SYSTEM FLASHER10_TEST (* Test FLASHER10 with D10U10B service interface *)
  (* Standard: 61499-1; Classification: Communication; Function: Test; Type: DeviceNet *)
  (* Version 0.0, 2003-05-01, JHC, Rockwell Automation, Modified from D10U10B_TEST *)
  DEVICE HMI : FRAME_DEVICE
    RESOURCE INS : PANEL_RESOURCE
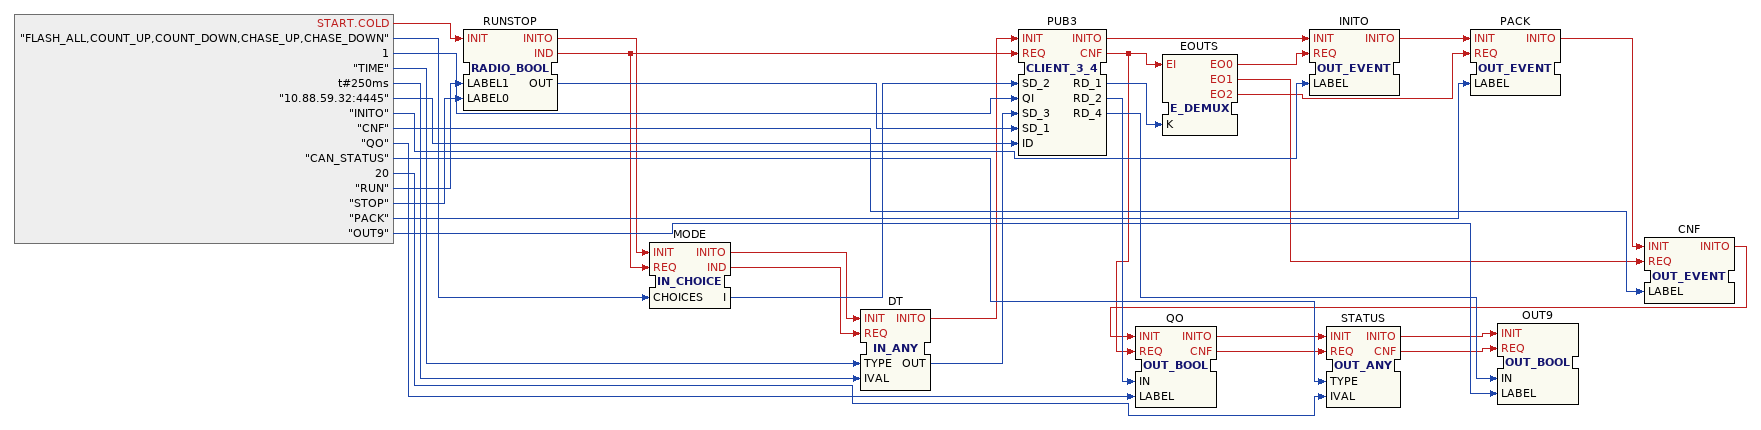
      FBS
        RUNSTOP : RADIO_BOOL;
        MODE : IN_CHOICE;
        DT : IN_ANY;
        PUB3 : CLIENT_3_4;
        EOUTS : E_DEMUX;
        INITO : OUT_EVENT;
        CNF : OUT_EVENT;
        QO : OUT_BOOL;
        STATUS : OUT_ANY;
        OUT9 : OUT_BOOL;
        PACK : OUT_EVENT;
      END_FBS
      EVENT_CONNECTIONS
        START.COLD TO RUNSTOP.INIT;
        RUNSTOP.INITO TO MODE.INIT;
        MODE.INITO TO DT.INIT;
        DT.INITO TO PUB3.INIT;
        PUB3.INITO TO INITO.INIT;
        INITO.INITO TO PACK.INIT;
        PACK.INITO TO CNF.INIT;
        CNF.INITO TO QO.INIT;
        QO.INITO TO STATUS.INIT;
        STATUS.INITO TO OUT9.INIT;
        RUNSTOP.IND TO MODE.REQ;
        MODE.IND TO DT.REQ;
        RUNSTOP.IND TO PUB3.REQ;
        PUB3.CNF TO QO.REQ;
        QO.CNF TO STATUS.REQ;
        STATUS.CNF TO OUT9.REQ;
        PUB3.CNF TO EOUTS.EI;
        EOUTS.EO0 TO INITO.REQ;
        EOUTS.EO1 TO CNF.REQ;
        EOUTS.EO2 TO PACK.REQ;
      END_CONNECTIONS
      DATA_CONNECTIONS
        MODE.I TO PUB3.SD_2;
        "FLASH_ALL,COUNT_UP,COUNT_DOWN,CHASE_UP,CHASE_DOWN" TO MODE.CHOICES;
        1 TO PUB3.QI;
        DT.OUT TO PUB3.SD_3;
        RUNSTOP.OUT TO PUB3.SD_1;
        PUB3.RD_1 TO EOUTS.K;
        PUB3.RD_2 TO QO.IN;
        PUB3.RD_4 TO OUT9.IN;
        "TIME" TO DT.TYPE;
        t#250ms TO DT.IVAL;
        "10.88.59.32:4445" TO PUB3.ID;
        "INITO" TO INITO.LABEL;
        "CNF" TO CNF.LABEL;
        "QO" TO QO.LABEL;
        "CAN_STATUS" TO STATUS.TYPE;
        20 TO STATUS.IVAL;
        "RUN" TO RUNSTOP.LABEL1;
        "STOP" TO RUNSTOP.LABEL0;
        "PACK" TO PACK.LABEL;
        "OUT9" TO OUT9.LABEL;
      END_CONNECTIONS
    END_RESOURCE
  END_DEVICE
  DEVICE CAN : CAN_DEV
    RESOURCE CTL : EMB_RES
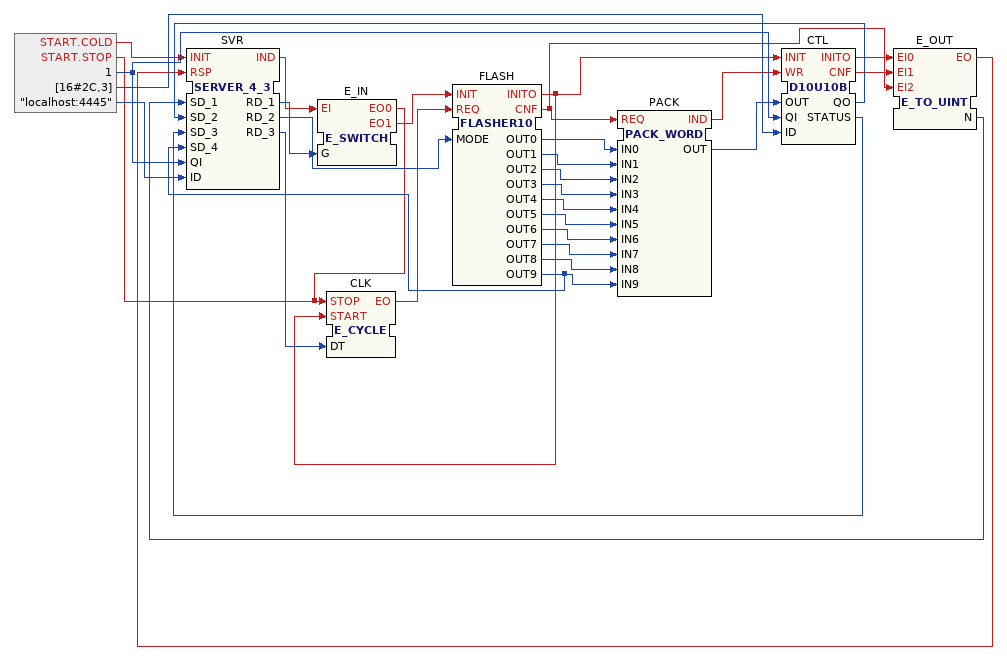
      FBS
        SVR : SERVER_4_3;
        E_IN : E_SWITCH;
        CLK : E_CYCLE;
        FLASH : FLASHER10;
        PACK : PACK_WORD;
        CTL : D10U10B;
        E_OUT : E_TO_UINT;
      END_FBS
      EVENT_CONNECTIONS
        START.COLD TO SVR.INIT;
        START.STOP TO CLK.STOP;
        SVR.IND TO E_IN.EI;
        E_IN.EO0 TO CLK.STOP;
        E_IN.EO1 TO FLASH.INIT;
        FLASH.INITO TO CTL.INIT;
        FLASH.INITO TO CLK.START;
        CLK.EO TO FLASH.REQ;
        FLASH.CNF TO PACK.REQ;
        PACK.IND TO CTL.WR;
        CTL.INITO TO E_OUT.EI0;
        CTL.CNF TO E_OUT.EI1;
        FLASH.CNF TO E_OUT.EI2;
        E_OUT.EO TO SVR.RSP;
      END_CONNECTIONS
      DATA_CONNECTIONS
        SVR.RD_1 TO E_IN.G;
        SVR.RD_2 TO FLASH.MODE;
        SVR.RD_3 TO CLK.DT;
        FLASH.OUT0 TO PACK.IN0;
        FLASH.OUT1 TO PACK.IN1;
        FLASH.OUT2 TO PACK.IN2;
        FLASH.OUT3 TO PACK.IN3;
        FLASH.OUT4 TO PACK.IN4;
        FLASH.OUT5 TO PACK.IN5;
        FLASH.OUT6 TO PACK.IN6;
        FLASH.OUT7 TO PACK.IN7;
        FLASH.OUT8 TO PACK.IN8;
        FLASH.OUT9 TO PACK.IN9;
        PACK.OUT TO CTL.OUT;
        E_OUT.N TO SVR.SD_1;
        CTL.QO TO SVR.SD_2;
        CTL.STATUS TO SVR.SD_3;
        FLASH.OUT9 TO SVR.SD_4;
        1 TO CTL.QI;
        1 TO SVR.QI;
        [16#2C,3] TO CTL.ID;
        "localhost:4445" TO SVR.ID;
      END_CONNECTIONS
    END_RESOURCE
    RESOURCE MGR : RMT_RES
    END_RESOURCE
  END_DEVICE
  DATA_CONNECTIONS (* parameter values *)
    [100,100,340,200] TO HMI.BOUNDS;
    [1,1] TO HMI.GRID;
    "10.88.59.32:61501" TO CAN.MGR_ID;
    0 TO CAN.FREQ;
  END_CONNECTIONS
END_SYSTEM
